// TIA Portal project "Conveyor Belt Process" (V16)

(* hardware
DEVICE "S7-1200 station_1"  S7-1200 Station
   slot 0: "Rack_0"  S7-1200 Rack  Rack  V1.0
   slot 1: "PLC_1"  CPU 1214C AC/DC/Rly  6ES7 214-1BG31-0XB0  V3.0
*)

// ===== PLC "PLC_1"  CPU 1214C AC/DC/Rly =====

VAR_GLOBAL   // PLC tag table "Default tag table"
   "Clock_Byte" AT %MB301 : Byte;
   "Clock_10Hz" AT %M301.0 : Bool;
   "Clock_5Hz" AT %M301.1 : Bool;
   "Clock_2.5Hz" AT %M301.2 : Bool;
   "Clock_2Hz" AT %M301.3 : Bool;
   "Clock_1.25Hz" AT %M301.4 : Bool;
   "Clock_1Hz" AT %M301.5 : Bool;
   "Clock_0.625Hz" AT %M301.6 : Bool;
   "Clock_0.5Hz" AT %M301.7 : Bool;
   "START BUTTON" AT %I0.0 : Bool;
   "STOP BUTTON" AT %I0.1 : Bool;
   "COUNTING SENSOR" AT %I0.2 : Bool;
   "ERROR DETECTOR" AT %I0.4 : Bool;
   "LIFE PROCESS" AT %Q0.0 : Bool;
   "CONVEYOR MOTOR" AT %Q0.1 : Bool;
   "ALARM - PRODUCT ERROR" AT %Q0.2 : Bool;
   "HMI START" AT %M0.0 : Bool;
   "HMI STOP" AT %M0.1 : Bool;
   "MARKER START" AT %M5.0 : Bool;
   "MARKER STOP" AT %M5.1 : Bool;
   "Tag_2" AT %M8.0 : Bool;
   "Tag_3" AT %IW64 : Int;
   "Tag_4" AT %MD100 : Real;
   "Tag_1" AT %M80.0 : Bool;
   "Tag_5" AT %MD200 : DWord;
   "Tag_6" AT %MD201 : DWord;
   "Tag_7" AT %MD300 : Time;
   "Tag_8" AT %M81.0 : Bool;
   "Tag_9" AT %M50.0 : Bool;
   "Tag_10" AT %M50.1 : Bool;
   "Tag_11" AT %MD20 : Time;
   "Tag_12" AT %MD24 : Time;
   "Tag_13" AT %M60.0 : Bool;
   "Tag_14" AT %M80.1 : Bool;
   "Tag_15" AT %MD203 : DWord;
   "Tag_16" AT %MD204 : DWord;
END_VAR

DATA_BLOCK "DATA_CONVEYOR"   // DB3
{ S7_Optimized_Access := 'FALSE' }
VERSION : 0.1
   VAR
      "PRODUCT COUNTER" : Int;
      "SPEED CONVEYOR" : Int;
      "VOLTAGE(V) CONVEYOR" : Real;
      "CURRENT(A) CONVEYOR" : Real;
   END_VAR
BEGIN
END_DATA_BLOCK

// folder: System blocks/Program resources

DATA_BLOCK "IEC_Counter_0_DB"   // DB1
{ S7_Optimized_Access := 'TRUE' }
AUTHOR : Simatic
FAMILY : IEC
NAME : CNTR
VERSION : 1.0
// stored: InstanceOfName IEC_COUNTER
"IEC_COUNTER"
BEGIN
END_DATA_BLOCK

DATA_BLOCK "IEC_Timer_0_DB"   // DB2
{ S7_Optimized_Access := 'TRUE' }
AUTHOR : Simatic
FAMILY : IEC
NAME : IEC_TMR
VERSION : 1.0
// stored: InstanceOfName IEC_TIMER
"IEC_TIMER"
BEGIN
END_DATA_BLOCK

DATA_BLOCK "IEC_Timer_0_DB_2"   // DB5
{ S7_Optimized_Access := 'TRUE' }
AUTHOR : Simatic
FAMILY : IEC
NAME : IEC_TMR
VERSION : 1.0
// stored: InstanceOfName IEC_TIMER
"IEC_TIMER"
BEGIN
END_DATA_BLOCK

// folder: (top level)

ORGANIZATION_BLOCK "Main"   // OB1, LAD, ProgramCycle
TITLE = "Main Program Sweep (Cycle)"
{ S7_Optimized_Access := 'TRUE' }
VERSION : 0.1
BEGIN

REGION Network 1
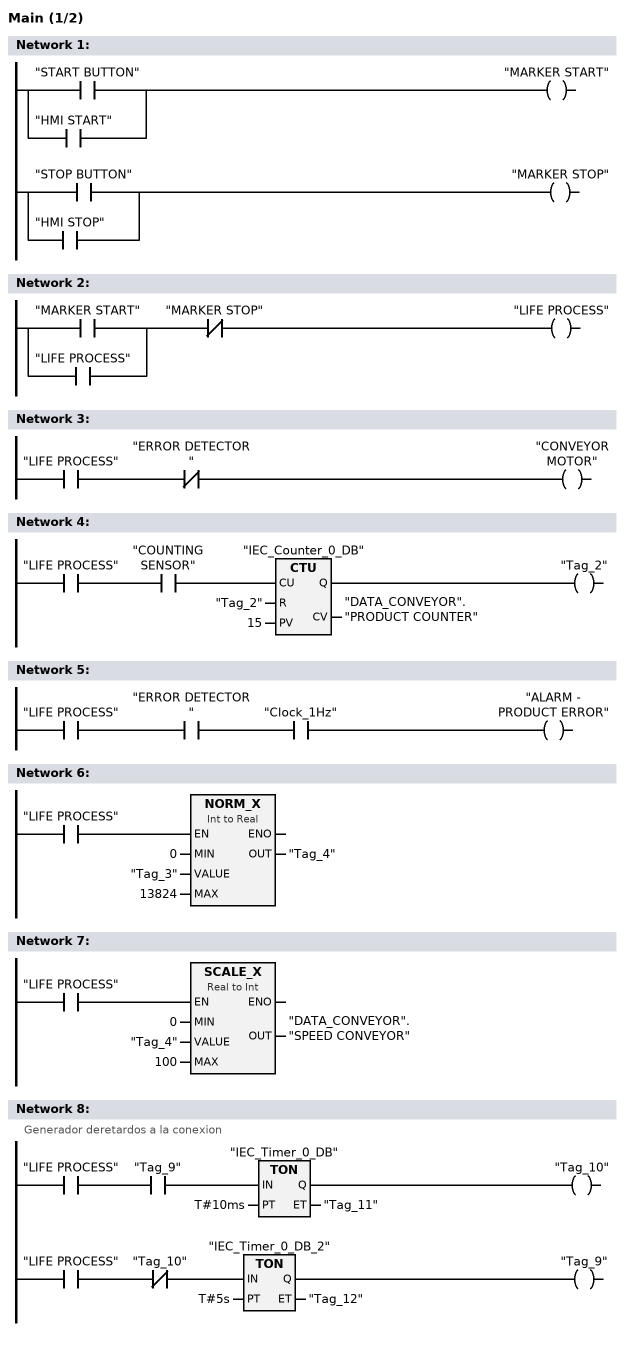
   RUNG wire#powerrail
      Contact( "START BUTTON" )
      wire#w1
      Coil( "MARKER START" )
   END_RUNG
   RUNG wire#powerrail
      Contact( "HMI START" )
   END_RUNG wire#w1
   RUNG wire#powerrail
      Contact( "STOP BUTTON" )
      wire#w2
      Coil( "MARKER STOP" )
   END_RUNG
   RUNG wire#powerrail
      Contact( "HMI STOP" )
   END_RUNG wire#w2
   // the same network as SCL:
   "MARKER START" := "START BUTTON" OR "HMI START";
   "MARKER STOP" := "STOP BUTTON" OR "HMI STOP";
END_REGION

REGION Network 2
   RUNG wire#powerrail
      Contact( "MARKER START" )
      wire#w1
      I_Contact( "MARKER STOP" )
      Coil( "LIFE PROCESS" )
   END_RUNG
   RUNG wire#powerrail
      Contact( "LIFE PROCESS" )
   END_RUNG wire#w1
   // the same network as SCL:
   "LIFE PROCESS" := ("MARKER START" OR "LIFE PROCESS") AND NOT "MARKER STOP";
END_REGION

REGION Network 3
   RUNG wire#powerrail
      Contact( "LIFE PROCESS" )
      I_Contact( "ERROR DETECTOR" )
      Coil( "CONVEYOR MOTOR" )
   END_RUNG
   // the same network as SCL:
   "CONVEYOR MOTOR" := "LIFE PROCESS" AND NOT "ERROR DETECTOR";
END_REGION

REGION Network 4
   "IEC_Counter_0_DB".CTU(CU := "LIFE PROCESS" AND "COUNTING SENSOR",
                          R := "Tag_2",
                          PV := 15,
                          CV => "DATA_CONVEYOR"."PRODUCT COUNTER");
   "Tag_2" := "IEC_Counter_0_DB".Q;
END_REGION

REGION Network 5
   RUNG wire#powerrail
      Contact( "LIFE PROCESS" )
      Contact( "ERROR DETECTOR" )
      Contact( "Clock_1Hz" )
      Coil( "ALARM - PRODUCT ERROR" )
   END_RUNG
   // the same network as SCL:
   "ALARM - PRODUCT ERROR" := "LIFE PROCESS" AND "ERROR DETECTOR" AND "Clock_1Hz";
END_REGION

REGION Network 6
   RUNG wire#powerrail
      Contact( "LIFE PROCESS" )
      { S7_Templates := "[SrcType := Int, DestType := Real]"; S7_GenerateENO := "TRUE" } Normalize(min := 0, value := "Tag_3", max := 13824, out => "Tag_4")
   END_RUNG
   // the same network as SCL:
   IF "LIFE PROCESS" THEN "Tag_4" := NORM_X(MIN := 0, VALUE := "Tag_3", MAX := 13824); END_IF;
END_REGION

REGION Network 7
   RUNG wire#powerrail
      Contact( "LIFE PROCESS" )
      { S7_Templates := "[SrcType := Real, DestType := Int]"; S7_GenerateENO := "TRUE" } Scale(min := 0, value := "Tag_4", max := 100, out => "DATA_CONVEYOR"."SPEED CONVEYOR")
   END_RUNG
   // the same network as SCL:
   IF "LIFE PROCESS" THEN
       "DATA_CONVEYOR"."SPEED CONVEYOR" := SCALE_X(MIN := 0, VALUE := "Tag_4", MAX := 100);
   END_IF;
END_REGION

REGION Network 8
   // Generador deretardos a la conexion
   "IEC_Timer_0_DB".TON(IN := "LIFE PROCESS" AND "Tag_9", PT := T#10ms, ET => "Tag_11");
   "Tag_10" := "IEC_Timer_0_DB".Q;
   "IEC_Timer_0_DB_2".TON(IN := "LIFE PROCESS" AND NOT "Tag_10", PT := T#5s, ET => "Tag_12");
   "Tag_9" := "IEC_Timer_0_DB_2".Q;
END_REGION

REGION Network 9
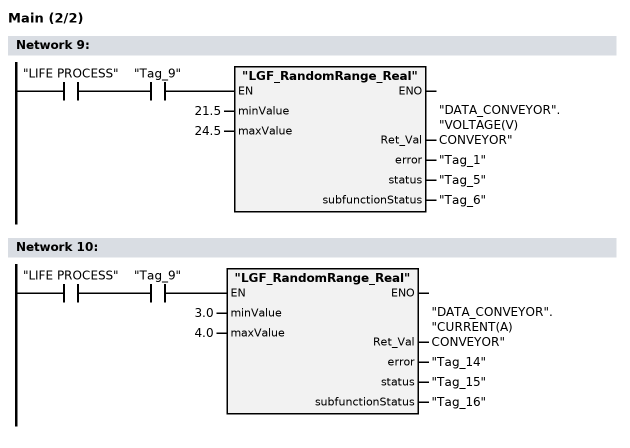
   RUNG wire#powerrail
      Contact( "LIFE PROCESS" )
      Contact( "Tag_9" )
      "LGF_RandomRange_Real"(minValue := 21.5, maxValue := 24.5, Ret_Val => "DATA_CONVEYOR"."VOLTAGE(V) CONVEYOR", error => "Tag_1", status => "Tag_5", subfunctionStatus => "Tag_6")
   END_RUNG
   // the same network as SCL:
   IF "LIFE PROCESS" AND "Tag_9" THEN
       "DATA_CONVEYOR"."VOLTAGE(V) CONVEYOR" := "LGF_RandomRange_Real"(minValue := 21.5,
                               maxValue := 24.5,
                               error => "Tag_1",
                               status => "Tag_5",
                               subfunctionStatus => "Tag_6");
   END_IF;
END_REGION

REGION Network 10
   RUNG wire#powerrail
      Contact( "LIFE PROCESS" )
      Contact( "Tag_9" )
      "LGF_RandomRange_Real"(minValue := 3.0, maxValue := 4.0, Ret_Val => "DATA_CONVEYOR"."CURRENT(A) CONVEYOR", error => "Tag_14", status => "Tag_15", subfunctionStatus => "Tag_16")
   END_RUNG
   // the same network as SCL:
   IF "LIFE PROCESS" AND "Tag_9" THEN
       "DATA_CONVEYOR"."CURRENT(A) CONVEYOR" := "LGF_RandomRange_Real"(minValue := 3.0,
                               maxValue := 4.0,
                               error => "Tag_14",
                               status => "Tag_15",
                               subfunctionStatus => "Tag_16");
   END_IF;
END_REGION
END_ORGANIZATION_BLOCK

// folder: LGF/4 Math operations

FUNCTION "LGF_RandomRange_Real" : Real   // FC10014, SCL
TITLE = LGF_RandomRange_Real
{ S7_Optimized_Access := 'TRUE' }
AUTHOR : Siemens_Digital_Industries
FAMILY : LGF
NAME : LGF_RandomRange_Real
// This function generates random numbers in defined limits (Datatype Real)
   VAR_INPUT
      minValue : Real;   // minimal Value random can reach / Minimum value of the range of the random number
      maxValue : Real;   // maximal Value random can reach / Maximum value of the range of the random number
   END_VAR
   VAR_OUTPUT
      error : Bool;   // Error if true
      status : Word;   // Status of the function
      subfunctionStatus : Word;   // Status or return value of called FB's, FCs and system blocks
   END_VAR
   VAR_TEMP
      tempTime : DTL;   // System time
      tempNanoSecondInDWord : DWord;   // UDINT converted to DWORD for access to individual bytes
      tempTimeStatus : Word;   // Status of the instruction RD_SYS_T
      tempRandomValue : DWord;   // Random-start-value
      tempNormReal : Real;   // normalized value
   END_VAR
   // Ret_Val : Returns random Real number in predefined range
   VAR CONSTANT
      ZERO : Real := 0.0;   // Zero value in case of error
      MAX_UDINT : UDInt := 4294967295;   // Maximum UDINT value
      SUB_STATUS_NO_ERROR : Word := 16#0000;   // Status: sub function call ends without error
      STATUS_FINISHED_NO_ERROR : Word := 16#0000;   // Status: Execution finished without errors
      ERR_MAX_LESS_MIN : Word := 16#8200;   // Error: The maximum limit number is smaller than the minimum limit number
      ERR_RD_SYS_T : Word := 16#8600;   // Error: System function Read system time returned an error
   END_VAR
BEGIN
   REGION Block info header
     //=============================================================================
     // SIEMENS AG / (c)Copyright 2017
     //-----------------------------------------------------------------------------
     // Title:            LGF_RandomRange_Real
     // Comment/Function: This function generates random numbers in defined limits (Datatype Real)
     // Library/Family:   LGF(Library General Functions)
     // Author:           Siemens Digital Industry Support
     // Tested with:      S7-PLCSIM Advanced V2.0 SP1
     // Engineering:      TIA Portal V15 Update 2
     // Restrictions:     ENO disabled - error handling done by error and status
     // Requirements:     PLC (S7-1200 / S7-1500)
     //-------------------------------------------------------------------------------
     // Change log table:
     // Version  | Date       | Expert in charge       | Changes applied
     //----------|------------|------------------------|------------------------------
     // 01.00.00 19.08.2015  Siemens Industry Online Support
     //                      First released version
     // 01.00.01 02.01.2017  Siemens Industry Online Support
     //                      Upgrade: TIA Portal V14 Update 1
     // 01.00.02 02.03.2017  Siemens Industry Online Support
     //                      Bugfix: FC number
     // 01.00.03 17.08.2018  Siemens Industry Online Support
     //                      Upgrade: TIA V15 Update 2
     // 01.00.04 23.11.2018  Siemens Industry Online Support
     //                      Upgrade: TIA V15.1
     // 01.01.00 13.11.2019  Siemens Industry Presales Support
     //                      Renamed from "LGF_RandomReal" to "LGF_RandomRange_Real"
     //                      Regions, commens and costants are added
     // 03.00.00 23.04.2020  Siemens Industry Support
     //                      Set version to V3.0.0, harmonize the version of the whole library
     //=============================================================================
   END_REGION

   REGION Validation
     // Check if the maximal Value is less than the minimal value
     IF (#minValue > #maxValue) THEN
       #error := true;
       #status := #ERR_MAX_LESS_MIN;
       #subfunctionStatus := #SUB_STATUS_NO_ERROR;
       #LGF_RandomRange_Real := #ZERO;
       RETURN;
     END_IF;

     // Read system time
     #tempTimeStatus := INT_TO_WORD(RD_SYS_T(#tempTime));

     // Check return variable for error
     IF (#tempTimeStatus <> #SUB_STATUS_NO_ERROR) THEN
       #error := true;
       #status := #ERR_RD_SYS_T;
       #subfunctionStatus := #tempTimeStatus;
       #LGF_RandomRange_Real := #ZERO;
       RETURN;
     END_IF;
   END_REGION

   REGION Calculating random number
     // Converting to double word so individual bytes can be addressed
     #tempNanoSecondInDWord := UDINT_TO_DWORD(#tempTime.NANOSECOND);

     // Calculate a random-start-value depending on the time
     #tempRandomValue.%B3 := #tempNanoSecondInDWord.%B0;
     #tempRandomValue.%B2 := #tempNanoSecondInDWord.%B1;
     #tempRandomValue.%B1 := #tempNanoSecondInDWord.%B2;
     #tempRandomValue.%B0 := #tempNanoSecondInDWord.%B3;

     // Norm the calculated random number: 0.0 <= #tempNormReal <= 1.0
     #tempNormReal := UDINT_TO_REAL(DWORD_TO_UDINT(#tempRandomValue)) / UDINT_TO_REAL(#MAX_UDINT);

     // Scale the tempNormReal to be in the range of maxValue and minValue
     #LGF_RandomRange_Real := ((#tempNormReal * (#maxValue - #minValue) + (#minValue)));

     #error := false;
     #status := #STATUS_FINISHED_NO_ERROR;
     #subfunctionStatus := #SUB_STATUS_NO_ERROR;
     // ENO mechanism is not used
     ENO := TRUE;
   END_REGION
END_FUNCTION